FUNCTION_BLOCK CROSSCOMM_SENDER_71FC4A2A5327CB09 (* Service Interface Function Block Type *)
  (* Standard: 61499-2 *)
  (* Version 0.0, 9/22/2017, bababen, nxtControl GmbH, template *)
  PACKAGE Main;
  (* Compiler Cpp nxtControl builtin 1.0 *)
  {SET_ATTRIBUTE(Runtime.FBType.ImplementingType, Runtime.System#DYNGEN_CROSSCOMM_SENDER)}
  {SET_ATTRIBUTE(Configuration.GenericFBType.InterfaceParams, Runtime.System#<InterfaceList> <EventInputs> <Event Name="CNF"> <With Var="LExtended" /> <With Var="LRetracted" /> </Event> </EventInputs> <InputVars> <VarDeclaration Name="LExtended" Type="BOOL" /> <VarDeclaration Name="LRetracted" Type="BOOL" /> </InputVars> </InterfaceList>)}
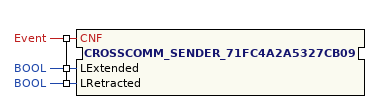
  EVENT_INPUT
    CNF WITH LExtended, LRetracted;
  END_EVENT
  VAR_INPUT
    LExtended : BOOL;
    LRetracted : BOOL;
  END_VAR
  EC_STATES
    START;
  END_STATES
END_FUNCTION_BLOCK
